// TwinCAT 3 PLC project LibraryVisionExample
// Title: LibraryVisionExample
// Company: Gema
// Author: RG
// ProjectVersion: 1.0.0.0
// ProgramVersion: 3.1.4024.0
// libraries:
//   LibraryVision, * (Gema)
//   Tc2_EtherCAT, * (Beckhoff Automation GmbH)
//   Tc2_Standard, * (Beckhoff Automation GmbH)
//   Tc2_System, * (Beckhoff Automation GmbH)
//   Tc2_TcpIp, * (Beckhoff Automation GmbH)
//   Tc3_Module, * (Beckhoff Automation GmbH)
//   TcoCore, 0.11.0.23 (Vortex.Library)
//   TcoData, 0.11.0.23 (Vortex.Library)
//   TcoDrivesBeckhoff, 0.11.0.23 (Vortex.Library)
//   TcoElements, 0.11.0.23 (Vortex.Library)
//   TcoIo, 0.11.0.23 (Vortex.Library)
//   TcoPneumatics, 0.11.0.23 (Vortex.Library)
// project tree:
//   CommRoboter/ ComRobo.TcPOU
//   CommRoboter/Struct/ ComRob.TcDUT, ComRobIn.TcDUT, ComRobOut.TcDUT, E_ConnectionSteps.TcDUT, FaultHandling.TcDUT, stTelegrammTCP.TcDUT, uTelegrammTCP.TcDUT
//   CommRoboter/Struct/Location/ Locations.TcDUT
//   ImplicitChecks/ CheckBounds.TcPOU, CheckRangeSigned.TcPOU, CheckRangeUnsigned.TcPOU
//   / PlcTask.TcTTO
//   POUs/ AppContext.TcPOU, MAIN.TcPOU, MainStation.TcPOU
// (motion and I/O tree: see PLC project libraryvision)
// real-time tasks:
//   TASK PlcTask: cycle T#1ms, priority 20, ADS port 350
// variable links:

CONFIGURATION LibraryVisionExample
    RESOURCE PLC ON TwinCAT3
        TASK PlcTask(INTERVAL := T#1ms, PRIORITY := 20);
        PROGRAM MAIN WITH PlcTask : MAIN;
    END_RESOURCE
END_CONFIGURATION

// ---- CommRoboter/Struct/ComRob.TcDUT
TYPE ComRob :
STRUCT
	//~
	in		: ComRobIn;
	out		: ComRobOut;
	//~
END_STRUCT
END_TYPE

// ---- CommRoboter/Struct/ComRobIn.TcDUT
TYPE
    ComRobIn :
    STRUCT
        {attribute addProperty Name "<#Station bereit fuer Spacer#>"}
        StationClearForSpacer : BOOL;
        {attribute addProperty Name "<#Home Pos erreicht#>"}
        HomePosReached : BOOL;
        {attribute addProperty Name "<#Fehler ID#>"}
        FaultID : INT;
        {attribute addProperty Name "<#Status Running#>"}
        StatusRunning : BOOL;
        {attribute addProperty Name "<#Fehler#>"}
        Fault : BOOL;
        {attribute addProperty Name "<#HighPower aktiv#>"}
        PowerOn : BOOL;
        {attribute addProperty Name "<#EStop aktiv#>"}
        Estop : BOOL;
        {attribute addProperty Name "<#Increase Index#"}
       IncreaseIndex: BOOL;
        {attribute addProperty Name "<#Index Palette Schaumstoffring#>"}
        PalletIndexPick : INT;
        {attribute addProperty Name "<#Berechneter Wert aus Roboter#>"}
        RowPallet : INT;
        {attribute addProperty Name "<#Foto machen#>"}
        TakeFoto : BOOL;
		   {attribute addProperty Name "<#Foto machen#>"}
        AnglePickOrigin : INT;
    END_STRUCT
END_TYPE

// ---- CommRoboter/Struct/ComRobOut.TcDUT
TYPE
    ComRobOut :
    STRUCT
        {attribute addProperty Name "<#AutoMode Aktiv#>"}
        ModeAuto        : BOOL;
        stopRun         : BOOL;
        reset           : BOOL;
        contactReady    : BOOL;
        contactPunched  : BOOL;
        homePosReq      : BOOL;
        tableInPos      : BOOL;
        HighPowerOn     : BOOL;
        PalletPickIndex : INT := 1;
        HighPowerOff    : BOOL;
        RowDone         : BOOL;
        //auf HMI: 
        //            - Toggle vor eindruecken der Kontakte
        //              - Hoehe einstellbar
        ContactHeight        : INT;
        WaitBeforeContacting : BOOL;
        {attribute addProperty Name "<#Foto Done#>"}
        FotoDone  : BOOL;
        Locations : Locations;
    END_STRUCT
END_TYPE

// ---- CommRoboter/Struct/E_ConnectionSteps.TcDUT
TYPE
    E_ConnectionSteps :
    (
        eCONNECTION_STATE_IDLE,
        eCONNECTION_STATE_CONNECT_START,
        eCONNECTION_STATE_CONNECT_WAIT,
        eCONNECTION_STATE_DATAEXCHANGE,
        eCONNECTION_STATE_CLOSE_START,
        eCONNECTION_STATE_CLOSE_WAIT,
        eCONNECTION_STATE_ERROR
    );
END_TYPE

// ---- CommRoboter/Struct/FaultHandling.TcDUT
TYPE
    FaultHandling :
    STRUCT
        FaultID : int;
    END_STRUCT
END_TYPE

// ---- CommRoboter/Struct/Location/Locations.TcDUT
TYPE
    Locations :
    STRUCT
        LocHeight : INT;
        LocWidth  : INT;
        Roll      : INT;
    END_STRUCT
END_TYPE

// ---- CommRoboter/Struct/stTelegrammTCP.TcDUT
{attribute 'pack_mode' := '1'}
TYPE
    stTelegrammTCP :
    STRUCT
        myStats  : ARRAY[1..4] OF BYTE;
        myInt    : ARRAY[1..8] OF INT;
        myBool   : ARRAY[1..12] OF INT;
        fillbyte : ARRAY[1..2] OF BYTE;
    END_STRUCT
END_TYPE

// ---- CommRoboter/Struct/uTelegrammTCP.TcDUT
TYPE uTelegrammTCP :
UNION
	//~
    stTel       : stTelegrammTCP;
    aTel        : ARRAY[1..SIZEOF(stTelegrammTCP)] OF BYTE;
    sTel        : STRING(SIZEOF(stTelegrammTCP));
	//~
END_UNION
END_TYPE

// ---- POUs/MAIN.TcPOU
PROGRAM MAIN
VAR
    _app : AppContext;
END_VAR

_app.Run();
_app.RtcSynchronize(true, '', 60);

END_PROGRAM

// ---- POUs/AppContext.TcPOU
FUNCTION_BLOCK AppContext EXTENDS TcoCore.TcoContext
VAR
    _mainStation : MainStation(THIS^);

    {attribute addProperty Name "Versionsnummer Plc"}
    _sVersion : STRING(23);
    //~
    _stProgramVersion : ST_LibVersion;
    //~

END_VAR

(*~
    <docu>
        <summary>
            Main method of the TcoContext. This is the entry point of any control logic that belongs to this context.
            The call of this method is ensured by calling the <c>InstanceName.Run()</c> method, and it must not be called explicitly.
            This method is abstract, and it must be overridden in derived block.
        </summary>
    </docu>
~*)
METHOD PROTECTED Main
_mainStation();

//IF (THIS^._startCycleCount MOD 10 = 0) THEN
//    Logger.Push('This is a log entry', eMessageCategory.Trace);
//END_IF;

//IF (THIS^._startCycleCount MOD 125 = 0) THEN
//    Logger.Push('This is a log entry', eMessageCategory.Info);
//END_IF;

//IF (THIS^._startCycleCount MOD 400 = 0) THEN
//    Logger.Push('This is a log entry', eMessageCategory.Warning);
//END_IF;

//IF (THIS^._startCycleCount MOD 2000 = 0) THEN
//    Logger.Push('This is a log entry', eMessageCategory.Error);
//END_IF;
END_METHOD

END_FUNCTION_BLOCK

// ---- POUs/MainStation.TcPOU
FUNCTION_BLOCK MainStation EXTENDS TcoCore.TcoObject
VAR
    counter : INT;

    _IvController            : LibraryVision.IVController(THIS^);
    _trigger                 : BOOL;
    _triggerR                : Tc2_Standard.R_TRIG;
    _coordinate              : BOOL;
    _coordinates             : ARRAY[0..2] OF LibraryVision.Coordinates;
    _distanceFromObject      : LREAL;
    _fieldOfView             : FieldOfView;
    _coordinatesInMillimeter : LREAL;
    _calculate               : BOOL;
END_VAR

VAR
	//~
    _comRob : ComRobo;

    _communicationStruct : ComRob;
    _msgToSend           : uTelegrammTCP;
    _msgReceive          : uTelegrammTCP;

    _arrayOfPositionValuesX                 : ARRAY[1..SIZE] OF INT;
    _arrayOfPositionValuesY                 : ARRAY[1..SIZE] OF INT;
    _arrayOfPositionValuesTheta             : ARRAY[1..SIZE] OF INT;
    _arrayOfPositionValuesInMillimeterX     : ARRAY[1..SIZE] OF INT;
    _arrayOfPositionValuesInMillimeterY     : ARRAY[1..SIZE] OF INT;
    _arrayOfPositionValuesInMillimeterTheta : ARRAY[1..SIZE] OF INT;
    _arrayOfCorrection                      : ARRAY[1..SIZE] OF ARRAY[ 0..2] OF INT;

    _index          : INT;
    _count          : INT;
    _aggrvValueX    : INT;
    _aggrevatedMidX : LREAL;
    _aggrvValueY    : INT;
    _aggrevatedMidY : LREAL;
	_increaseIndex : Tc2_Standard.R_TRIG	;
	//~
END_VAR
VAR CONSTANT
    SIZE           : INT  := 30;
    SIZE_OF_PALLET : INT := 27; // 9 reihen, 3 columns
END_VAR

counter := counter + 1;
_increaseIndex(clk := _communicationStruct.in.IncreaseIndex);

IF (THIS^.counter MOD 13 = 0) THEN
    THIS^.Messenger.Info('opalalla').Pin();
END_IF

IF (THIS^.counter MOD 400 = 0) THEN
    THIS^.Messenger.Error('ich Poste').Pin();
END_IF

_IvController();

_triggerR(clk := _communicationStruct.in.TakeFoto);

IF _triggerR.Q THEN
    _trigger := TRUE;
END_IF

IF NOT _communicationStruct.in.TakeFoto THEN
    _communicationStruct.out.FotoDone := FALSE;
END_IF

IF _trigger THEN
    IF _IvController.TriggerSensorMethod().Done THEN
        _trigger    := FALSE;
        _coordinate := TRUE;

    end_if
END_IF

IF _coordinate THEN
    IF _IvController.ReadTool1CoordinatesMethod().Done
           and _IvController.ReadTool2CoordinatesMethod().Done
           and _IvController.ReadTool3CoordinatesMethod().Done THEN
        _coordinate     := FALSE;
        _coordinates[0] := _IvController.RawCoordinatesTool1;
        _coordinates[1] := _IvController.RawCoordinatesTool2;
        _coordinates[2] := _IvController.RawCoordinatesTool3;

        _arrayOfPositionValuesX[_communicationStruct.out.PalletPickIndex]     := DINT_TO_INT(_coordinates[0].xValue);
        _arrayOfPositionValuesY[_communicationStruct.out.PalletPickIndex]     := DINT_TO_INT(_coordinates[0].yValue);
        _arrayOfPositionValuesTheta[_communicationStruct.out.PalletPickIndex] :=
            DINT_TO_INT(_coordinates[0].variableValue);

        _calculate := TRUE;
    END_IF
END_IF

IF _calculate THEN
    IF _IvController.CalculationMethod().Done THEN
        _calculate          := FALSE;
        _distanceFromObject := _IvController.CalculationTask.DistanceFromObject;
        _fieldOfView        := _IvController.CalculationTask.FieldOfView;

        _arrayOfPositionValuesInMillimeterX[_communicationStruct.out.PalletPickIndex] :=
            DINT_TO_INT(_IvController.CalculationTask.CoordinatesInMillimeter.xValue);

        _arrayOfPositionValuesInMillimeterY[_communicationStruct.out.PalletPickIndex] :=
            DINT_TO_INT(_IvController.CalculationTask.CoordinatesInMillimeter.yValue);

        _arrayOfPositionValuesInMillimeterTheta[_communicationStruct.out.PalletPickIndex] :=
            DINT_TO_INT(_IvController.CalculationTask.CoordinatesInMillimeter.variableValue);

        _aggrevatedMidX := _aggrvValueX / _count;
        _aggrevatedMidY := _aggrvValueY / _count;

        _communicationStruct.out.PalletPickIndex := 1;

    END_IF

    IF _increaseIndex.q THEN
        _communicationStruct.out.PalletPickIndex := _communicationStruct.out.PalletPickIndex + 1;

        IF _communicationStruct.out.PalletPickIndex > SIZE_OF_PALLET THEN

            //            FOR _index := 1 TO SIZE_OF_PALLET DO
            //                IF _arrayOfPositionValuesInMillimeterX[_index] <> 0 THEN
            //                    _aggrvValueX := _aggrvValueX + _arrayOfPositionValuesInMillimeterX[_index];
            //                    _aggrvValueY := _aggrvValueY + _arrayOfPositionValuesInMillimeterY[_index];
            //                    _count       := _count + 1;
            //                END_IF
            //            END_FOR
			_communicationStruct.out.PalletPickIndex := 1;
        END_IF

        _communicationStruct.out.FotoDone := TRUE;
        PositionCorrectionFactor();
        //        IF  _communicationStruct.in.RowPallet <> 0 THEN

    END_IF

END_IF

RunCommunication();

METHOD PRIVATE MapComRob : BOOL
VAR_INST
    _start :BOOL;
    n : INT;

    _powerOn : BOOL;
    _powerOnTr : Tc2_Standard.R_TRIG;
    _powerOffTr : Tc2_Standard.R_TRIG;
    sigTimer : Tc2_Standard.TON;
    sigTime : TIME := T#1000MS;
END_VAR
//TCP IP Komm
////==========in
_communicationStruct.in.TakeFoto := INT_TO_BOOL(_msgReceive.stTel.myBool[1]);
//_communicationStruct.in.Fault             := INT_TO_BOOL(_msgReceive.stTel.myBool[2]);
//_communicationStruct.in.HomePosReached    := INT_TO_BOOL(_msgReceive.stTel.myBool[3]);
_communicationStruct.in.IncreaseIndex        := INT_TO_BOOL(_msgReceive.stTel.myBool[4]);
//_communicationStruct.in.StatusRunning     := INT_TO_BOOL(_msgReceive.stTel.myBool[5]);
//_communicationStruct.in.PowerOn           := INT_TO_BOOL(_msgReceive.stTel.myBool[6]);
//_communicationStruct.in.Estop             := INT_TO_BOOL(_msgReceive.stTel.myBool[7]);
//_communicationStruct.in.ContactGrasped    := INT_TO_BOOL(_msgReceive.stTel.myBool[8]);
//_communicationStruct.in.SectionClearTable := INT_TO_BOOL(_msgReceive.stTel.myBool[9]);
//_communicationStruct.in.CoilDone          := INT_TO_BOOL(_msgReceive.stTel.myBool[10]);
_communicationStruct.in.PalletIndexPick := _msgReceive.stTel.myInt[1];
_communicationStruct.in.RowPallet       := _msgReceive.stTel.myInt[2];
_communicationStruct.in.AnglePickOrigin := _msgReceive.stTel.myInt[3];
///==================== OUT
//_msgToSend.stTel.myBool[1]  := BOOL_TO_INT(_communicationStruct.out.ModeAuto);
//_msgToSend.stTel.myBool[2]  := BOOL_TO_INT(_communicationStruct.out.stopRun);
//_msgToSend.stTel.myBool[3]  := BOOL_TO_INT(_communicationStruct.out.reset);
//_msgToSend.stTel.myBool[4]  := BOOL_TO_INT(_communicationStruct.out.contactReady);
//_msgToSend.stTel.myBool[5]  := BOOL_TO_INT(_communicationStruct.out.contactPunched);
//_msgToSend.stTel.myBool[6]  := BOOL_TO_INT(_communicationStruct.out.homePosReq);
//_msgToSend.stTel.myBool[7]  := BOOL_TO_INT(_communicationStruct.out.tableInPos);
//_msgToSend.stTel.myBool[8]  := BOOL_TO_INT(_communicationStruct.out.HighPowerOn);
//_msgToSend.stTel.myBool[9]  := BOOL_TO_INT(_communicationStruct.out.HighPowerOff);
//_msgToSend.stTel.myBool[11] := BOOL_TO_INT(_communicationStruct.out.RowDone);

_msgToSend.stTel.myBool[10] := BOOL_TO_INT(_communicationStruct.out.FotoDone);
_msgToSend.stTel.myInt[1]   := _communicationStruct.out.PalletPickIndex;
_msgToSend.stTel.myInt[3] := _communicationStruct.out.Locations.LocHeight;
_msgToSend.stTel.myInt[4] := _communicationStruct.out.Locations.LocWidth;
_msgToSend.stTel.myInt[5] := _communicationStruct.out.Locations.Roll;

//TEsten, start darf nur einmal ausgeführt werden
IF _start THEN
    _start := FALSE;
    n      := n + 1;
END_IF
END_METHOD

METHOD PositionCorrectionFactor : BOOL
VAR_INST
	// Werte experimentiell mit Versuchen ermittelt
    averageValueX     : INT := 299;
    averageValueY     : INT := 286;
    averageValueRoll : INT:= 0;
	_index : INT;
	
	anglePickOrigin : REAL ;
END_VAR
_index := _communicationStruct.out.PalletPickIndex - 1;

// Umrechhung in RealWert, WinkelWert fuer Korrektur notwendig
anglePickOrigin :=  _communicationStruct.in.AnglePickOrigin/ 10;

IF THIS^._IvController.ID01StatusProp.Total_Status_OK THEN
    _communicationStruct.out.Locations.LocWidth :=
      averageValueX -   THIS^._arrayOfPositionValuesInMillimeterX[_index];

    _communicationStruct.out.Locations.LocHeight :=
      averageValueY -   THIS^._arrayOfPositionValuesInMillimeterY[_index] ;

    _communicationStruct.out.Locations.Roll :=
        averageValueRoll - THIS^._arrayOfPositionValuesInMillimeterTheta[_index];
ELSE
    _communicationStruct.out.Locations.LocHeight := 0;
    _communicationStruct.out.Locations.LocWidth  := 0;
    _communicationStruct.out.Locations.Roll      := 0;
END_IF

_arrayOfCorrection[_index][0] := _communicationStruct.out.Locations.LocHeight;
_arrayOfCorrection[_index][1] := _communicationStruct.out.Locations.LocWidth;
_arrayOfCorrection[_index][2] := _communicationStruct.out.Locations.Roll;
END_METHOD

METHOD PRIVATE RunCommunication
 _comRob(_msgSend:= _msgToSend, _msgRcv:= _msgReceive);
 
 MapComRob();
END_METHOD

END_FUNCTION_BLOCK

// ---- CommRoboter/ComRobo.TcPOU
FUNCTION_BLOCK ComRobo
VAR_IN_OUT
    _msgSend : uTelegrammTCP;
    _msgRcv  : uTelegrammTCP;
END_VAR
VAR
    _sRemoteHost     : STRING            := '192.168.3.208';
    _serverPort      : UDINT             := 7000;
    eStep            : E_ConnectionSteps := E_ConnectionSteps.eCONNECTION_STATE_IDLE;
    _bEnable         : BOOL              := TRUE;
    _comTrig         : Tc2_Standard.f_TRIG;
    _comStatus       : BOOL;
    _bConnected      : BOOL;
    _bDisconnect     : BOOL;
    fbServerCon      : Tc2_TcpIp.FB_ClientServerConnection;
    fbSend           : Tc2_TcpIp.FB_SocketSend;
    fbRceive         : Tc2_TcpIp.FB_SocketReceive;
    cbLen            : UDINT;
    bExecute         : BOOL;
    tTimeout         : TIME                    := T#2S;
    eState           : E_SocketConnectionState := eSOCKET_DISCONNECTED;
    sSrvNetId        : T_AmsNetId              := '';
    hSocket          : T_HSOCKET;
    bExecuteRec      : BOOL;
    bBusy            : BOOL;
    bError           : BOOL;
    nErrId           : UDINT;
    nRecBytes        : UDINT;
    _hbOld           : INT := 0;
    _hb              : INT;
    _hbErrCoun       : INT;
    index            : uINT;
    _reset           : BOOL;
    fbPollTimer      : Tc2_Standard.TON := (PT := TIME#10MS); (* Receive poll timer *)
    fbReconnectTimer : Tc2_Standard.TON := (pt := TIME#1S);
    fbResponseTimer  : Tc2_Standard.TON := (pt := TIME#160MS); (* Response timeout timer *)
    fbTimeOut        : Tc2_Standard.TON := (pt := TIME#2S);    //Time OUt für ANtwort
    reconnectTime    : TIME             := T#1S;
    _index           : INT              := 0;
    _dataRcv         : Tc2_Standard.R_TRIG;
    _bConnectedTrig  : Tc2_Standard.R_TRIG;
    _n               : INT;
    _ErrorCycle      : UDINT;
    faultID          : FaultHandling;
END_VAR
VAR CONSTANT
    hbError : INT := 5;
END_VAR


IF NOT _bConnected THEN
    mClearData();
END_IF

IF _comTrig.Q THEN
    //    fbReconnectTimer(pt := T#0MS);
    IF _comStatus THEN
        _comStatus := FALSE;
        _bEnable   := FALSE;
    ELSE
        _bEnable   := TRUE;
        _comStatus := true;
    END_IF

    //else
    //    fbReconnectTimer(pt := t#5s);
END_IF

//StateMachine f+ür die TCP/IP Com
//Solange Enable true, versucht der Baustein eine Verbindung aufzubauen
//Gesamte Zeitüberwachung für bEnable und keine Verbindung, -> als Error an HMI
fbPollTimer(in := NOT fbPollTimer.Q);
fbResponseTimer(in := NOT fbResponseTimer.Q);

CASE eStep OF
    eCONNECTION_STATE_IDLE:
        IF _bEnable XOR _bConnected THEN
            IF _bEnable THEN
                fbReconnectTimer(in := TRUE);

                IF fbReconnectTimer.Q THEN
                    _bDisconnect := FALSE;
                    nRecBytes    := 0;
                    fbReconnectTimer(in := FALSE, pt := reconnectTime);
                    estep := eCONNECTION_STATE_CONNECT_START;
                END_IF
            ELSE
                estep := eCONNECTION_STATE_CLOSE_START;
            END_IF
        ELSIF _bConnected THEN
            estep := eCONNECTION_STATE_DATAEXCHANGE;
        ELSE
            fbReconnectTimer(in := FALSE);
        END_IF
    eCONNECTION_STATE_CONNECT_START:
        cbLen := SIZEOF(_msgSend.aTel) + 1;
        //Rücksetzten Heartbeat
        _hb        := 0;
        _hbOld     := 0;
        _hbErrCoun := 0;

        fbServerCon
        (
            sSrvNetID     :=
            , nMode       := Tc2_TcpIp.CONNECT_MODE_ENABLEDBG
            , sRemoteHost := _sRemoteHost
            , nRemotePort := _serverPort
            , bEnable     := _bEnable
            , tReconnect  := reconnectTime
            , bBusy       => bBusy
            , bError      => bError
            , nErrId      => nErrId
            , hSocket     => hSocket
            , eState      => eState
        );

        IF NOT fbServerCon.bBusy THEN
            IF NOT fbServerCon.bError THEN
                _n := _n + 1;

                IF _n >= 2 THEN
                    _n          := 0;
                    _bConnected := TRUE;

                    Tc2_System.ADSLOGSTR
                    (
                        msgCtrlMask := Tc2_System.ADSLOG_MSGTYPE_WARN
                        , msgFmtStr := 'Connection via TCP/IP established mit %s! '
                        , strArg    := 'Omron Rob'
                    );

                    faultID.FaultID := 0;
                END_IF

                eStep := eCONNECTION_STATE_IDLE;
            ELSE
                Tc2_System.ADSLOGSTR
                (
                    msgCtrlMask := Tc2_System.ADSLOG_MSGTYPE_WARN
                    , msgFmtStr := 'fbServerCon geht nicht %s'
                    , strArg    := UDINT_TO_STRING(fbServerCon.nErrId)
                );

                // Fehler, dass die Connection nicht zustande kommt fürs HMI
                // Lösung vermutlihc, Omron Comm-Programm muss neugestartet werden,
                // da ein Heartbeat FEhler vorliegt
                _bConnectedTrig(clk := _bConnected);
                faultID.FaultID := 10;
                eStep           := eCONNECTION_STATE_ERROR;
                _n              := 0;
            END_IF
        END_IF
    eCONNECTION_STATE_DATAEXCHANGE:
        _bDisconnect := NOT _bEnable OR _bDisconnect; //(kann aufs Hmi gelegt werden

        IF _bDisconnect AND NOT (fbSend.bBusy OR fbRceive.bBusy) THEN
            _bDisconnect := FALSE;
            eStep        := eCONNECTION_STATE_CLOSE_START;
        ELSE
            //Sender der Daten
            IF NOT (_bDisconnect OR fbSend.bBusy) THEN
                IF fbResponseTimer.q AND NOT fbRceive.bBusy THEN
                    fbSend(bExecute := FALSE);

                    fbSend
                    (
                        sSrvNetId  := sSrvNetId
                        , hSocket  := fbServerCon.hSocket
                        , cbLen    := cbLen
                        , pSrc     := ADR(_msgSend.aTel)
                        , bExecute := TRUE
                        , tTimeout := tTimeout
                        , bBusy    => bBusy
                        , bError   => bError
                        , nErrId   => nErrId
                    );
                END_IF
            ELSE
                fbSend(bExecute := FALSE);

                IF fbSend.bError THEN
                    Tc2_System.ADSLOGSTR
                    (
                        msgCtrlMask := Tc2_System.ADSLOG_MSGTYPE_WARN
                        , msgFmtStr := 'fbSend %s'
                        , strArg    := UDINT_TO_STRING(fbServerCon.nErrId)
                    );
                END_IF
            END_IF

            //===================Recieve Data =================================
            IF NOT (_bDisconnect OR fbRceive.bBusy) THEN
                IF fbPollTimer.Q THEN
                    fbRceive(bExecute := FALSE);

                    fbRceive
                    (
                        sSrvNetId   := sSrvNetId
                        , hSocket   := fbServerCon.hSocket
                        , cbLen     := cbLen
                        , pDest     := ADR(_msgRcv.aTel)
                        , bExecute  := TRUE
                        , tTimeout  := tTimeout
                        , bBusy     => bBusy
                        , bError    => bError
                        , nErrId    => nErrId
                        , nRecBytes =>
                    );

                    // CHekcehn des HEartbeats, ob Änderungen da sind
                    _hb := BYTE_TO_INT(_msgRcv.stTel.myStats[3]);
                    fbRceive(nRecBytes => nRecBytes);

                    IF _hb = _hbOld THEN
                        fbTimeOut(in := TRUE);
                    ELSE
                        fbTimeOut(in := false);
                    END_IF

                    IF nRecBytes <> 0 THEN
                        IF _hb = _hbOld THEN
                            _hbErrCoun := _hbErrCoun + 1;

                            IF _hbErrCoun > 2 THEN
                                _ErrorCycle := _ErrorCycle + 1;
                            end_if
                        ELSIF _hb <> _hbOld OR _hb = 0 THEN
                            _hbErrCoun                := 0;
                            _msgSend.stTel.myStats[3] := INT_TO_BYTE(_hb);
                        END_IF
                    END_IF

                    //===========================================================
                    //=========================================================
                    IF _hbErrCoun > hbError OR fbTimeOut.q THEN
                        _bDisconnect := TRUE;

                        //                        //                        mClearData();
                        FOR index := 1 TO UDINT_TO_UINT(cbLen) DO
                            _msgRcv.aTel[index] := 0;
                        END_FOR

                        Tc2_System.ADSLOGSTR
                        (
                            msgCtrlMask := Tc2_System.ADSLOG_MSGTYPE_WARN
                            , msgFmtStr := 'HEartBeat Fehler, Verbindung verloren'
                            , strArg    := ''
                        );
                    END_IF

                    _hbOld := _hb;
                END_IF
            ELSE
                fbRceive(bExecute := FALSE);

                IF NOT fbRceive.bError THEN
                    //watchdog von Omron, "HEartBeat"
                    //                    _msgSend.stTel.myStats[5] := _msgRcv.stTel.myStats[5];
                ELSE
                    _bDisconnect := TRUE;

                    Tc2_System.ADSLOGSTR
                    (
                        msgCtrlMask := Tc2_System.ADSLOG_MSGTYPE_WARN
                        , msgFmtStr := 'fbSocketRec %s'
                        , strArg    := UDINT_TO_STRING(fbRceive.nErrId)
                    );
                END_IF
            END_IF
        END_IF
    eCONNECTION_STATE_CLOSE_START:
        Tc2_System.ADSLOGSTR
        (
            msgCtrlMask := Tc2_System.ADSLOG_MSGTYPE_WARN
            , msgFmtStr := 'Verbindung mit Omron wird geschlossen'
            , strArg    := ''
        );

        fbServerCon(bEnable := FALSE);
        fbTimeOut(in := FALSE);

        IF NOT fbServerCon.bBusy THEN
            _bConnected := FALSE;

            IF NOT fbServerCon.bError THEN
                eStep := eCONNECTION_STATE_IDLE;
            ELSE
                Tc2_System.ADSLOGSTR
                (
                    msgCtrlMask := Tc2_System.ADSLOG_MSGTYPE_WARN
                    , msgFmtStr := 'fbSocketClose %s'
                    , strArg    := UDINT_TO_STRING(fbServerCon.nErrId)
                );

                eStep := eCONNECTION_STATE_ERROR;
            END_IF
        END_IF
    eCONNECTION_STATE_ERROR: (* Error step *)
        IF _bConnected THEN
            eStep := eCONNECTION_STATE_CLOSE_START;
        ELSE
            eStep := eCONNECTION_STATE_IDLE;
        END_IF
END_CASE

METHOD PRIVATE mClearData : BOOL
VAR
    _index : UINT;
END_VAR
// The warning can be disabled here as the user is aware of the risk that the reference may not be valid by checking its validity
{warning disable C0371}
IF NOT __ISVALIDREF(_msgRcv) THEN
    RETURN;
END_IF

FOR _index := 1 TO SIZEOF(_msgRcv) - 1 DO
    _msgRcv.aTel[_index] := 0;
END_FOR

// The warning may be restored at the end of the access area
{warning restore C0371}
END_METHOD

METHOD PRIVATE mTestComCauseOfErr : BOOL
VAR_INST
    i     : INT;
    fbTon : Tc2_Standard.TON;
END_VAR
//wird später gelöscht

////Dient dem TEst, warum die Verbindung manchmal abbricht
//fbTon(in := NOT fbTon.Q, pt := T#500MS);

//IF fbton.Q THEN
//    FOR i := 1 TO 12 DO
//        IF gIOs._msgSend.stTel.myBool[i] THEN
//            gIOs._msgSend.stTel.myBool[i] := 0;
//        ELSE
//            gIOs._msgSend.stTel.myBool[i] := 1;
//        END_IF
//    END_FOR

//FOR i := 1 TO 8 DO
//    IF gIOs._msgSend.stTel.myBool[i] THEN
//        gIOs._msgSend.stTel.myInt[i] := gIOs._msgSend.stTel.myInt[i] + 1;

//    END_IF
//END_FOR

//END_IF
END_METHOD

END_FUNCTION_BLOCK

// ---- ImplicitChecks/CheckBounds.TcPOU
// Implicitly generated code : DO NOT EDIT
FUNCTION CheckBounds : DINT
VAR_INPUT
    index, lower, upper : DINT;
END_VAR

// Implicitly generated code : Only an Implementation suggestion
{noflow}
IF index < lower THEN
    CheckBounds := lower;
ELSIF index > upper THEN
    CheckBounds := upper;
ELSE
    CheckBounds := index;
END_IF

{flow}

END_FUNCTION

// ---- ImplicitChecks/CheckRangeSigned.TcPOU
// Implicitly generated code : DO NOT EDIT
FUNCTION CheckRangeSigned : DINT
VAR_INPUT
    value, lower, upper : DINT;
END_VAR

// Implicitly generated code : Only an Implementation suggestion
{noflow}
IF (value < lower) THEN
    CheckRangeSigned := lower;
ELSIF (value > upper) THEN
    CheckRangeSigned := upper;
ELSE
    CheckRangeSigned := value;
END_IF

{flow}

END_FUNCTION

// ---- ImplicitChecks/CheckRangeUnsigned.TcPOU
// Implicitly generated code : DO NOT EDIT
FUNCTION CheckRangeUnsigned : UDINT
VAR_INPUT
    value, lower, upper : UDINT;
END_VAR

// Implicitly generated code : Only an Implementation suggestion
{noflow}
IF (value < lower) THEN
    CheckRangeUnsigned := lower;
ELSIF (value > upper) THEN
    CheckRangeUnsigned := upper;
ELSE
    CheckRangeUnsigned := value;
END_IF

{flow}

END_FUNCTION
